// TIA Portal project "simbaaa" (V16)

(* hardware
DEVICE "HMI_1"  KTP700 Basic DP
   slot 0: "HMI_1"  KTP700 Basic DP  6AV2 123-2GA03-0AX0  16.0.0.0
   slot 1: "HMI_RT_1"  KTP700 Basic DP  6AV2 123-2GA03-0AX0  16.0.0.0
   slot 7: "HMI_1.MPI/DP_CP_1"  MPI/DP Interface  16.0.0.0
DEVICE "S7300/ET200M station_1"  S7-300 station
   slot 0: "Rail_0"  Rail  6ES7 390-1***0-0AA0
   slot 2: "PLC_1"  CPU 314C-2 DP  6ES7 314-6CH04-0AB0  V3.3
      slot 0: "MPI interface_1"  MPI
      slot 1: "DP interface_1"  DP
      slot 2: "DI 24/DO 16_1"  DI24/DO16
      slot 3: "AI 5/AO 2_1"  AI5/AO2
      slot 4: "Count_1"  Counter
      slot 5: "Positioning_1"  Positioning
*)

// ===== PLC "PLC_1"  CPU 314C-2 DP =====

VAR_GLOBAL   // PLC tag table "Default tag table"
   "Start" AT %M0.0 : Bool;
   "Stop" AT %M0.1 : Bool;
   "packets sensor" AT %M0.2 : Bool;
   "conveyer 1" AT %Q0.0 : Bool;
   "conveyer 2" AT %Q0.1 : Bool;
   "conveyer 3" AT %Q0.2 : Bool;
   "oil heater timer" AT %T0 : Timer;
   "frying" AT %Q0.3 : Bool;
   "counter" AT %C0 : Counter;
   "chip fryer timer" AT %T1 : Timer;
   "loading timer" AT %T2 : Timer;
   "cutting" AT %Q0.4 : Bool;
   "temperature sensor" AT %QW2 : Int;
   "counter output" AT %QW4 : Int;
   "conveyer 4" AT %Q0.5 : Bool;
   "restart" AT %Q0.6 : Bool;
   "oil heating" AT %Q0.7 : Bool;
   "bags sensor" AT %M0.3 : Bool;
   "truck" AT %Q1.0 : Bool;
END_VAR

ORGANIZATION_BLOCK "Main"   // OB1, LAD
TITLE = "Main Program Sweep (Cycle)"
{ S7_Optimized_Access := 'FALSE' }
VERSION : 0.1
   VAR_TEMP
      OB1_EV_CLASS : Byte;   // Bits 0-3 = 1 (Coming event), Bits 4-7 = 1 (Event class 1)
      OB1_SCAN_1 : Byte;   // 1 (Cold restart scan 1 of OB 1), 3 (Scan 2-n of OB 1)
      OB1_PRIORITY : Byte;   // Priority of OB Execution
      OB1_OB_NUMBR : Byte;   // 1 (Organization block 1, OB1)
      OB1_RESERVED_1 : Byte;   // Reserved for system
      OB1_RESERVED_2 : Byte;   // Reserved for system
      OB1_PREV_CYCLE : Int;   // Cycle time of previous OB1 scan (milliseconds)
      OB1_MIN_CYCLE : Int;   // Minimum cycle time of OB1 (milliseconds)
      OB1_MAX_CYCLE : Int;   // Maximum cycle time of OB1 (milliseconds)
      OB1_DATE_TIME : Date_And_Time;   // Date and time OB1 started
   END_VAR
   VAR_TEMP   // added for the SCL form of the ladder/FBD networks
      _w1 : Bool;
      _s5time1 : S5Time;
   END_VAR
BEGIN

REGION Network 1
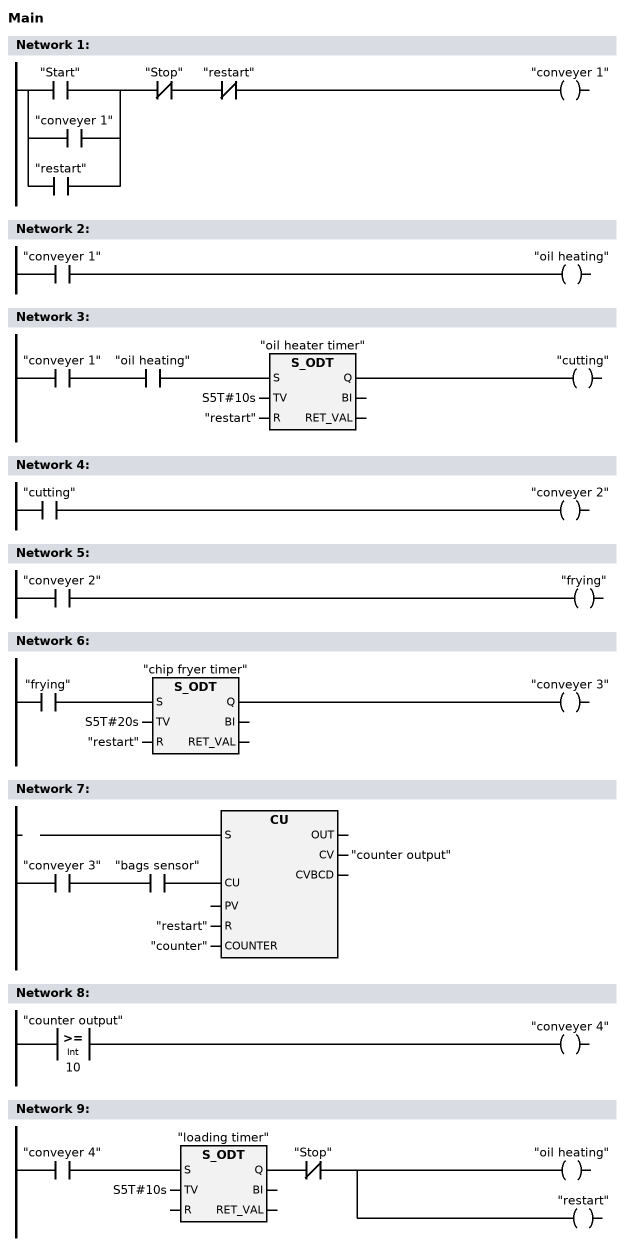
   RUNG wire#powerrail
      Contact( "Start" )
      wire#w1
      I_Contact( "Stop" )
      I_Contact( "restart" )
      Coil( "conveyer 1" )
   END_RUNG
   RUNG wire#powerrail
      Contact( "conveyer 1" )
   END_RUNG wire#w1
   RUNG wire#powerrail
      Contact( "restart" )
   END_RUNG wire#w1
   // the same network as SCL:
   "conveyer 1" := ("Start" OR "conveyer 1" OR "restart") AND NOT "Stop" AND NOT "restart";
END_REGION

REGION Network 2
   RUNG wire#powerrail
      Contact( "conveyer 1" )
      Coil( "oil heating" )
   END_RUNG
   // the same network as SCL:
   "oil heating" := "conveyer 1";
END_REGION

REGION Network 3
   RUNG wire#powerrail
      Contact( "conveyer 1" )
      Contact( "oil heating" )
      S_ODT(T_NO := "oil heater timer", TV := S5T#10s, R := "restart", BI =>, RET_VAL =>)
      Coil( "cutting" )
   END_RUNG
   // the same network as SCL:
   #_s5time1 := S_ODT(T_NO := "oil heater timer",
                      S := "conveyer 1" AND "oil heating",
                      TV := S5T#10s,
                      R := "restart",
                      Q => #_w1);
   "cutting" := #_w1;
END_REGION

REGION Network 4
   RUNG wire#powerrail
      Contact( "cutting" )
      Coil( "conveyer 2" )
   END_RUNG
   // the same network as SCL:
   "conveyer 2" := "cutting";
END_REGION

REGION Network 5
   RUNG wire#powerrail
      Contact( "conveyer 2" )
      Coil( "frying" )
   END_RUNG
   // the same network as SCL:
   "frying" := "conveyer 2";
END_REGION

REGION Network 6
   RUNG wire#powerrail
      Contact( "frying" )
      S_ODT(T_NO := "chip fryer timer", TV := S5T#20s, R := "restart", BI =>, RET_VAL =>)
      Coil( "conveyer 3" )
   END_RUNG
   // the same network as SCL:
   #_s5time1 := S_ODT(T_NO := "chip fryer timer", S := "frying", TV := S5T#20s, R := "restart", Q => #_w1);
   "conveyer 3" := #_w1;
END_REGION

REGION Network 7
   // no SCL statement known for Cu: written as a call
   Cu(cu := "conveyer 3" AND "bags sensor", r := "restart", "counter" := "counter", cv => "counter output");
END_REGION

REGION Network 8
   RUNG wire#powerrail
      { S7_Templates := "SrcType := Int" } GE_Contact(in1 := "counter output", in2 := 10)
      Coil( "conveyer 4" )
   END_RUNG
   // the same network as SCL:
   "conveyer 4" := "counter output" >= 10;
END_REGION

REGION Network 9
   RUNG wire#powerrail
      Contact( "conveyer 4" )
      S_ODT(T_NO := "loading timer", TV := S5T#10s, R :=, BI =>, RET_VAL =>)
      I_Contact( "Stop" )
      wire#w1
      Coil( "oil heating" )
   END_RUNG
   RUNG wire#w1
      Coil( "restart" )
   END_RUNG
   // the same network as SCL:
   #_s5time1 := S_ODT(T_NO := "loading timer", S := "conveyer 4", TV := S5T#10s, Q => #_w1);
   "oil heating" := #_w1 AND NOT "Stop";
   "restart" := "oil heating";
END_REGION
END_ORGANIZATION_BLOCK

(* ===== HMI "HMI_RT_1" =====
system functions are stored by id; their names below are inferred from use
connection "HMI_Connection_1": IF1 B, SIMATIC S7 300/400 MPI

HMI tags "Default tag table"
   "Tag_ScreenNumber" : UInt, internal
   "move" : Int, internal
   "conveyer 4" : Bool = PLC "conveyer 4" AT %Q0.5, 1 s
   "counter output" : Int = PLC "counter output" AT %QW4, 1 s
   "conveyer 1" : Bool = PLC "conveyer 1" AT %Q0.0, 1 s
   "Start" : Bool = PLC Start AT %M0.0, 1 s
   "Stop" : Bool = PLC Stop AT %M0.1, 1 s
   "conveyer 2" : Bool = PLC "conveyer 2" AT %Q0.1, 1 s
   "conveyer 3" : Bool = PLC "conveyer 3" AT %Q0.2, 1 s
   "moving things" : Int, internal
   "HM" : Int, internal

Template "Template_1" 800x480
   Button "Exit" at 714,429 size 71x50; TextOff 'Exit'; PictureOff "ExitRuntime_KTP700_Basic_DP_TR"; PictureOn "ExitRuntime_KTP700_Basic_DP_TR"
      on Release: StopRuntime(0)
   Button "Template_Button" at 614,429 size 71x50; TextOff 'Text'
   Button "Template_Button_1" at 514,429 size 71x50; TextOff 'Text'
   Button "Template_Button_2" at 414,429 size 71x50; TextOff 'Text'
   Button "Template_Button_3" at 314,429 size 71x50; TextOff 'Text'
   Button "Template_Button_4" at 214,429 size 71x50; TextOff 'Text'
   Button "Alarms" at 114,429 size 71x50; TextOff 'Alarms'; PictureOff "AlarmDisplay_KTP700_Basic_DP_TR"; PictureOn "AlarmDisplay_KTP700_Basic_DP_TR"
      on Release: function_ef3f5d25("Alarm window_Unacknowledged", -1)
   Button "Start screen" at 14,429 size 71x50; TextOff 'Start screen'; PictureOff "NavigateHome_KTP700_Basic_DP_TR"; PictureOn "NavigateHome_KTP700_Basic_DP_TR"
      on Release: ActivateScreen("Root screen", 0)
   SymbolicIOField "Symbolic_IO_Field_Screen" at 93,9 size 600x33; TextOff '0'; TextOn '1'; TextList "TextList_ScreenNames"
      ProcessValue <- "Tag_ScreenNumber"
      on Change: ActivateScreenByNumber("Tag_ScreenNumber", 0)
   DateTimeField "HmiScreenItemData" at 695,25 size 105x25
   DateTimeField "HmiScreenItemData_1" at 695,0 size 105x25
   GraphicView "Logo" at 0,0 size 91x51; Picture "Logo of HMI_1"

screen "Root screen" 800x480, template "Template_1"
   on GenerateScreen: SetTag("Tag_ScreenNumber", 1); function_f9c01323("move", 1, 100, 0, 1); function_f9c01323("moving things", 1, 100, 0, 1); function_f9c01323("HM", 1, 100, 0, 1)
   Button "Button_1" at 16,48 size 96x32; TextOff 'Start'
      on Press: SetBit("Start"); ActivateScreen("Screen_1", 0)
      on Release: ResetBit("Start")
   Button "Button_2" at 127,48 size 96x32; TextOff 'Stop'
      on Release: ResetBit("Stop")
      on Press: SetBit("Stop")
   IOField "I/O field_1" at 648,109 size 96x32; FormatPattern s99999
      ProcessValue <- "counter output"
   Button "Button_3" at 630,64 size 145x32; TextOff 'counting bags'
   GraphicView "Graphic view_1" at 443,225 size 29x50; Picture "Graphic_1"
   GraphicView "Graphic view_2" at 455,390 size 58x33; Picture "Graphic_2"
   GraphicView "Graphic view_3" at 6,218 size 38x29; Picture "Graphic_2"
      HorizontalMovement <- "moving things"
      Visibility <- "conveyer 1"
   GraphicView "Graphic view_4" at 154,284 size 39x29; Picture "Graphic_2"
      HorizontalMovement <- "HM"
   GraphicView "Graphic view_5" at 300,350 size 32x31; Picture "Graphic_2"
   GraphicView "Graphic view_6" at 0,188 size 185x29; Picture "Graphic_3"
   GraphicView "Graphic view_7" at 142,244 size 190x36; Picture "Graphic_3"
   GraphicView "Graphic view_8" at 443,347 size 181x40; Picture "Graphic_3"
   GraphicView "Graphic view_9" at 286,306 size 202x35; Picture "Graphic_3"
   GraphicView "Graphic view_10" at 605,280 size 195x148; Picture "Graphic_5"
   GraphicView "Graphic view_11" at 30,164 size 44x31; Picture "DM_20241004035037_001"
      HorizontalMovement <- "move"
      Visibility <- "conveyer 1"
   GraphicView "Graphic view_12" at 163,225 size 47x36; Picture "downloa]d"
      HorizontalMovement <- "move"
      Visibility <- "conveyer 2"
   GraphicView "Graphic view_13" at 316,273 size 46x50; Picture "download"
      Visibility <- "conveyer 3"
      HorizontalMovement <- "move"
   GraphicView "Graphic view_14" at 464,317 size 56x52; Picture "Graphic_6"
      HorizontalMovement <- "move"
      Visibility <- "conveyer 4"
   GraphicView "Graphic view_16" at 122,160 size 42x34; Picture "Graphic_8"
   GraphicView "Graphic view_15" at 276,205 size 40x55; Picture "Graphic_9"

screen "Screen_1" 800x480
   Button "Button_1" at 8,8 size 96x32; TextOff 'Text'
      on Press: function_efd93a16()
*)